FUNCTION Convert_TOD_TO_REAL : Hresult
VAR_INPUT
	in : TOD;
	out : REFERENCE TO REAL;
END_VAR
VAR
	converted : REAL;
END_VAR
VAR CONSTANT
	INCOMPATIBLE : HRESULT := 16#9811070E;
END_VAR

converted := TOD_TO_REAL(in);

IF (REAL_TO_TOD(converted) <> in) THEN
	Convert_TOD_TO_REAL := INCOMPATIBLE;
	RETURN;
END_IF

out := converted;

END_FUNCTION

(* stored: Version 1.1.0.1, ProductVersion 3.1.4024.12
   POU Convert_TOD_TO_REAL: Id {798b73de-22ca-4fbe-b89c-1910de451198}, SpecialFunc None *)
